# EPICS substitutions: iocBoot/ioc6idACS1/substitutions/pseudoMotor.substitutions
# Pseudo-motors
# Note: This databases will be in the next release of motor, not in 6idACS1App

# This is a simple example using the sumDiff2D database.  This takes 2 real motors and makes 2 soft motors,
# SUM which moves both motors together, and DIFF which moves them in opposite directions.
# It can be used for slits, for K/B mirror benders, etc.

file "$(MOTOR)/motorApp/Db/pseudoMotor.db"
{
pattern
{M,           DINP,                        OUT,                     RDBL,                          STOO,     DESC, EGU, DIR, VELO, VBAS, ACCL, BDST, BVEL,                    BACC, MRES,   RRES, PREC,  DHLM, DLLM}
{pm1, "6idACS1:KBV:Done NPP NMS", "6idACS1:pm1DVAL.VAL PP MS", "6idACS1:KBV:Readback.G NPP NMS", "6idACS1:KBV:Stop PP MS",    "Vert. curvature",          mm,  Pos,   1,    .1,   .1,    0,    1,   .1, .1,     1.0,  3,    10000, -10000}
{pm2, "6idACS1:KBV:Done NPP NMS", "6idACS1:pm2DVAL.VAL PP MS", "6idACS1:KBV:Readback.H NPP NMS", "6idACS1:KBV:Stop PP MS",    "Vert. Ellipticity",        mm,  Pos,   1,    .1,   .1,    0,    1,   .1, .1,     1.0,  3,    10000, -10000}
{pm3, "6idACS1:KBH:Done NPP NMS", "6idACS1:pm3DVAL.VAL PP MS", "6idACS1:KBH:Readback.G NPP NMS", "6idACS1:KBH:Stop PP MS",    "Hor. curvature",          mm,  Pos,   1,    .1,   .1,    0,    1,   .1, .1,     1.0,  3,    10000, -10000}
{pm4, "6idACS1:KBH:Done NPP NMS", "6idACS1:pm4DVAL.VAL PP MS", "6idACS1:KBH:Readback.H NPP NMS", "6idACS1:KBH:Stop PP MS",    "Hor. ellipticity",        mm,  Pos,   1,    .1,   .1,    0,    1,   .1, .1,     1.0,  3,    10000, -10000}
}

file "$(MOTOR)/motorApp/Db/sumDiff2D.db"
{
pattern
{T,   SUM, DIFF,      M1DRV,     M1RBV,    M2DRV,    M2RBV,    M1STOP,    M1DONE,    M2STOP,    M2DONE,  PREC}
{KBV:,  pm1,  pm2,    m17.VAL,   m17.RBV,  m18.VAL,  m18.RBV,  m17.STOP,  m17.DMOV,  m18.STOP,  m18.DMOV,    1}
{KBH:,  pm3,  pm4,    m19.VAL,   m19.RBV,  m20.VAL,  m20.RBV,  m19.STOP,  m19.DMOV,  m20.STOP,  m20.DMOV,    1}
}
